// TIA Portal V21 export
TYPE "UDT_WORK_CNT"
   STRUCT
      S : USInt;
      "M" : USInt;
      H : UDInt;
   END_STRUCT;
END_TYPE
